ABB RobotStudio station: Robot_1.rsstnx

Station Robot_1 (saved by RobotStudio 22.3.10190.2)
Controller 14M_63302, task T_ROB1: task frame (RAPID world) sits at (0, 0, 955) mm in the station
Controller 14M_63302
  mechanical unit ROB_1: IRB140_6_81_C_03, 6 joints, base frame (0, 0, 0) mm
Layout (positions relative to the parent item):
  - IRB140_6_81_C_03 [mechanism, from Robots\IRB140_6_81_C_G_03.rslib] at (0, 0, 955) mm; joint values [0, 0, 0, 0, 0.5236, 0] (rad or m)
  - base [part, from Herramienta\base.rslib] at (-69.84, 0, 0) mm
  - pinza [mechanism, from Herramienta\pinza.rslib] at (506.29, 0, 1634.5) mm, rotated rx 180 ry 60 rz 180 deg
Attachment: pinza is attached to IRB140_6_81_C_03 / Link6
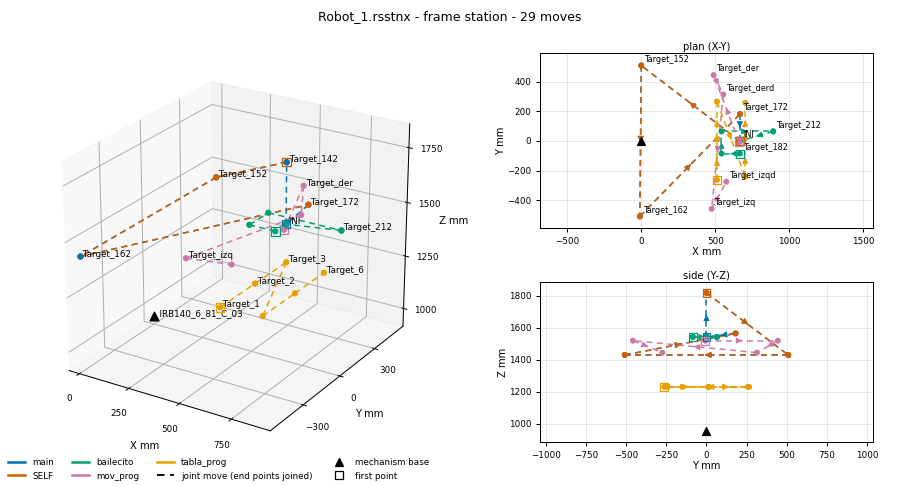
[picture p0: tool path of Robot_1.rsstnx in frame station, 29 of 29 moves have a stored position in this frame; points joined in program order, loops and branches not executed]
Targets, tools, work objects and paths stored in the station, written as RAPID:
! task T_ROB1
MODULE CalibData
  PERS tooldata pinza:=[TRUE,[[0,0,184],[1,0,0,0]],[0.8,[0,0,1],[1,0,0,0],0,0,0]];
  TASK PERS wobjdata INICIO:=[FALSE,TRUE,"",[[0,0,100],[1,0,0,0]],[[0,0,0],[1,0,0,0]]];
  TASK PERS wobjdata TOOL_INI:=[FALSE,TRUE,"",[[0,0,100],[1,0,0,0]],[[0,0,0],[1,0,0,0]]];
  TASK PERS wobjdata selfie:=[FALSE,TRUE,"",[[0,0,0],[1,0,0,0]],[[0,0,0],[1,0,0,0]]];
  TASK PERS wobjdata baile:=[FALSE,TRUE,"",[[0,0,0],[1,0,0,0]],[[0,0,0],[1,0,0,0]]];
  TASK PERS wobjdata prog:=[FALSE,TRUE,"",[[0,0,0],[1,0,0,0]],[[0,0,0],[1,0,0,0]]];
  TASK PERS wobjdata tabla:=[FALSE,TRUE,"",[[0,0,0],[1,0,0,0]],[[0,0,0],[1,0,0,0]]];
ENDMODULE

! task T_ROB1
MODULE Module1
  CONST robtarget INI:=[[665.640325542,0,487.5],[0.5,0,0.866025404,0],[0,0,0,0],[9E+09,9E+09,9E+09,9E+09,9E+09,9E+09]];
  CONST robtarget Target_142:=[[665.64041018,0,861.837012818],[0.499999994,0,0.866025407,0],[0,0,0,0],[9E+09,9E+09,9E+09,9E+09,9E+09,9E+09]];
  CONST robtarget Target_152:=[[-0.963032928,509.640010522,475.218174883],[0.080203662,-0.703189698,0.701874156,0.080400809],[1,0,-1,0],[9E+09,9E+09,9E+09,9E+09,9E+09,9E+09]];
  CONST robtarget Target_162:=[[-10.300026127,-509.536826166,475.218174883],[0.079509613,0.709601869,0.695390732,-0.081087231],[-2,0,-1,0],[9E+09,9E+09,9E+09,9E+09,9E+09,9E+09]];
  CONST robtarget Target_172:=[[665.640420298,181.047016927,609.643692497],[0.500000017,0.000000006,0.866025394,0.000000032],[0,-1,0,0],[9E+09,9E+09,9E+09,9E+09,9E+09,9E+09]];
  CONST robtarget INI_TOOL:=[[506.291630361,0.000000055,684.334688154],[0.016951444,0.003304092,-0.999833129,-0.005953702],[-1,0,-1,0],[9E+09,9E+09,9E+09,9E+09,9E+09,9E+09]];
  CONST robtarget Target_182:=[[665.640420098,-85.360458869,587.499963629],[0.500000009,0,0.866025398,-0.000000007],[-1,0,-1,0],[9E+09,9E+09,9E+09,9E+09,9E+09,9E+09]];
  CONST robtarget Target_192:=[[541.099087196,-85.360454561,587.499966997],[0.500000008,0,0.866025399,0.000000002],[-1,0,-1,0],[9E+09,9E+09,9E+09,9E+09,9E+09,9E+09]];
  CONST robtarget Target_202:=[[541.099082331,64.503649199,587.499967763],[0.500000014,0.000000002,0.866025396,0.000000004],[0,-1,0,0],[9E+09,9E+09,9E+09,9E+09,9E+09,9E+09]];
  CONST robtarget Target_212:=[[890.204075016,64.503647282,587.4999638],[0.50000001,0.000000002,0.866025398,0.000000004],[0,-1,0,0],[9E+09,9E+09,9E+09,9E+09,9E+09,9E+09]];
  CONST robtarget Target_222:=[[890.204069077,64.503618601,587.500000402],[0.573032675,0.225673257,0.76972677,-0.168005456],[0,1,-2,1],[9E+09,9E+09,9E+09,9E+09,9E+09,9E+09]];
  CONST robtarget cablat:=[[665.640421771,-0.00000793,587.49996474],[0.479991416,0.140029407,0.831369522,0.242538089],[-1,0,-1,0],[9E+09,9E+09,9E+09,9E+09,9E+09,9E+09]];
  CONST robtarget cablat2:=[[665.640420566,-0.000009406,587.499964594],[0.484065894,-0.125220713,0.838426714,-0.216888515],[0,-1,0,0],[9E+09,9E+09,9E+09,9E+09,9E+09,9E+09]];
  CONST robtarget Target_izq:=[[474.535955149,-459.198261849,564.393522923],[0.447769621,0.328423296,0.811674085,-0.181178601],[-1,0,-1,0],[9E+09,9E+09,9E+09,9E+09,9E+09,9E+09]];
  CONST robtarget Target_der:=[[487.932313273,444.93760695,564.393522923],[0.450404663,-0.316362197,0.816450636,0.174524952],[0,-1,0,0],[9E+09,9E+09,9E+09,9E+09,9E+09,9E+09]];
  CONST robtarget Target_cen:=[[660.297702447,-7.372961274,564.393522923],[0.483027998,0.004888302,0.875587109,-0.002696689],[-1,0,0,0],[9E+09,9E+09,9E+09,9E+09,9E+09,9E+09]];
  CONST robtarget Target_izqd:=[[573.869959953,-275.294847407,489.780166033],[0.415074942,0.200687881,0.882340173,-0.094408612],[-1,-1,0,0],[9E+09,9E+09,9E+09,9E+09,9E+09,9E+09]];
  CONST robtarget Target_derd:=[[553.589537064,314.090127827,489.780166033],[0.411582805,-0.230912076,0.874916807,0.108626831],[0,-1,-1,0],[9E+09,9E+09,9E+09,9E+09,9E+09,9E+09]];
  CONST robtarget Target_1:=[[510.581971914,-262.52385287,276.40159081],[0.071314829,-0.234598663,-0.969319224,-0.017259911],[-1,0,0,0],[9E+09,9E+09,9E+09,9E+09,9E+09,9E+09]];
  CONST robtarget Target_6:=[[701.720701408,257.984497295,276.401631453],[0.071390696,0.230297295,-0.970350166,0.016943449],[0,-1,-1,0],[9E+09,9E+09,9E+09,9E+09,9E+09,9E+09]];
  CONST robtarget Target_5:=[[701.720735215,16.842353635,276.401584514],[0.07139064,0.230297311,-0.970350166,0.01694347],[0,-1,-1,0],[9E+09,9E+09,9E+09,9E+09,9E+09,9E+09]];
  CONST robtarget Target_4:=[[701.720733974,-241.16510292,276.401596915],[0.071390537,0.23029737,-0.970350158,0.016943509],[-1,-1,-1,0],[9E+09,9E+09,9E+09,9E+09,9E+09,9E+09]];
  CONST robtarget Target_2:=[[510.581967502,10.186684173,276.401598409],[0.071314778,-0.234598704,-0.969319217,-0.017259947],[-1,0,0,0],[9E+09,9E+09,9E+09,9E+09,9E+09,9E+09]];
  CONST robtarget Target_3:=[[510.581960996,266.120914072,276.401597862],[0.071314801,-0.234598704,-0.969319215,-0.017259948],[0,0,0,0],[9E+09,9E+09,9E+09,9E+09,9E+09,9E+09]];
  PROC main()
    MoveJ INI,v1000,z100,pinza\WObj:=INICIO;
    bailecito;
    WaitTime 2;
    MoveJ Target_142,v1000,fine,pinza\WObj:=selfie;
    WaitTime 2;
    MoveJ Target_152,v1000,fine,pinza\WObj:=selfie;
    WaitTime 2;
    MoveJ Target_162,v1000,fine,pinza\WObj:=selfie;
    WaitTime 2;
    MoveJ Target_172,v1000,fine,pinza\WObj:=selfie;
    WaitTime 2;
    MoveJ INI,v1000,z100,pinza\WObj:=INICIO;
  ENDPROC
  PROC SELF()
    MoveJ Target_142,v1000,fine,pinza\WObj:=selfie;
    MoveJ Target_152,v1000,fine,pinza\WObj:=selfie;
    MoveJ Target_162,v1000,fine,pinza\WObj:=selfie;
    MoveJ Target_172,v1000,fine,pinza\WObj:=selfie;
  ENDPROC
  PROC bailecito()
    MoveJ Target_182,v300,fine,pinza\WObj:=baile;
    MoveJ Target_192,v300,fine,pinza\WObj:=baile;
    MoveJ Target_202,v300,fine,pinza\WObj:=baile;
    MoveJ Target_212,v300,fine,pinza\WObj:=baile;
    MoveJ Target_222,v300,fine,pinza\WObj:=baile;
    MoveJ cablat,v300,fine,pinza\WObj:=baile;
    MoveJ cablat2,v300,fine,pinza\WObj:=baile;
    MoveJ INI,v300,fine,pinza\WObj:=INICIO;
  ENDPROC
  PROC mov_prog()
    MoveJ Target_cen,v1000,fine,pinza\WObj:=prog;
    MoveJ Target_der,v1000,fine,pinza\WObj:=prog;
    MoveJ Target_derd,v1000,fine,pinza\WObj:=prog;
    MoveJ Target_izq,v1000,fine,pinza\WObj:=prog;
    MoveJ Target_izqd,v1000,fine,pinza\WObj:=prog;
  ENDPROC
  PROC tabla_prog()
    MoveJ Target_1,v1000,fine,pinza\WObj:=tabla;
    MoveJ Target_2,v1000,fine,pinza\WObj:=tabla;
    MoveJ Target_3,v1000,fine,pinza\WObj:=tabla;
    MoveJ Target_4,v1000,fine,pinza\WObj:=tabla;
    MoveJ Target_5,v1000,fine,pinza\WObj:=tabla;
    MoveJ Target_6,v1000,fine,pinza\WObj:=tabla;
  ENDPROC
ENDMODULE

